TYPE DUT_NCI_Steuern :
STRUCT
	Pfad				: STRING := 'C:\SRTvisu\Fräsanlage\GCodes\';
	PrgName				: STRING := '';
	Override			: DINT;
	Reset				: BOOL;
	Koppeln				: BOOL;
	Start				: BOOL;
	StopOverrideNull	: BOOL;
	EinzelsatzStart		: BOOL;
	EinzelsatzWeiter	: BOOL;	
END_STRUCT
END_TYPE

(* stored: Version 1.1.0.1
   DUT DUT_NCI_Steuern: Id {7f1f5931-274a-49eb-910f-844b7d2e2467} *)
